FUNCTION_BLOCK FB_ModeManager
VAR_INPUT
	xEStop: BOOL;
	xSel_Auto: BOOL;
	xSel_Manual: BOOL;
END_VAR
VAR_OUTPUT
	eMode: E_MODE;
	eErrorType: E_ErrorHAndling;
END_VAR
VAR
	fbErrorHandling: FB_ErrorHAndling;
END_VAR

IF IOs.xMC_HasError OR xEStop THEN  //Emergency_Stop is NC designed!
	eMode:= Error;
  ELSIF IOs.xSel_Auto THEN
   eMode:= Auto;
	ELSIF IOs.xSel_Manual THEN
		eMode:= Manual;
		ELSE
			eMode:= Idle;
END_IF


fbErrorHandling(xEStop := xEStop);
eErrorType:= fbErrorHandling.eErrorHandling;

END_FUNCTION_BLOCK

(* stored: Version 1.1.0.1
   POU FB_ModeManager: Id {3a909d5a-4d8d-4531-aacf-bcb8147f0a11}, SpecialFunc None *)
